// SIMATIC S7-200 SMART project (STEP 7-Micro/WIN SMART), CPU ST40

ORGANIZATION_BLOCK MAIN:OB1
TITLE=程序注释
BEGIN
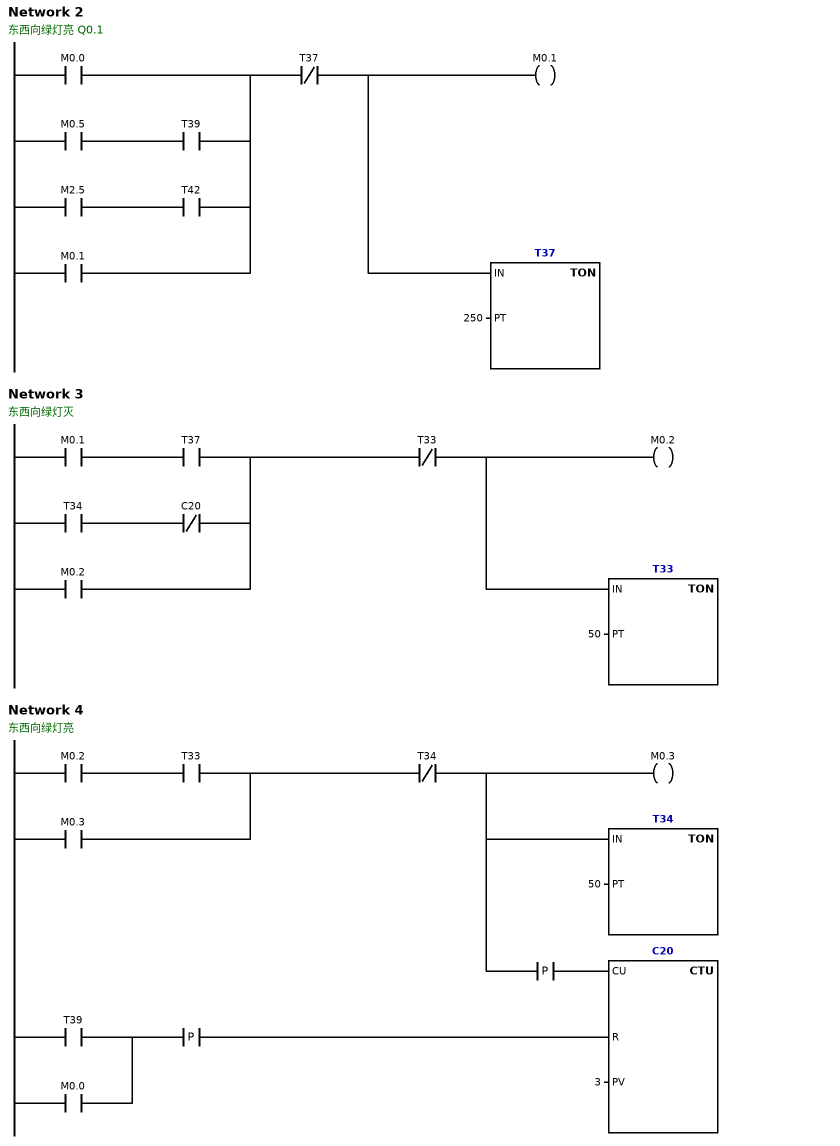
Network 2
// 东西向绿灯亮 Q0.1
// (network saved uncompiled; LAD cells follow)
// row 0: c0 -| |- M0.0  c1 -- v  c2 -|/|- T37 v  c3 --  c4 -( ) M0.1
// row 1: c0 -| |- M0.5  c1 -| |- T39 ^v  c2 ^v
// row 2: c0 -| |- M2.5  c1 -| |- T42 ^v  c2 ^v
// row 3: c0 -| |- M0.1  c1 -- ^  c2 ^  c3 --  c4 [TON T37 IN:=power@row3, PT:=250]
// row 4: c4 [box]
Network 3
// 东西向绿灯灭
// (network saved uncompiled; LAD cells follow)
// row 0: c0 -| |- M0.1  c1 -| |- T37 v  c2 --  c3 -|/|- T33 v  c4 --  c5 -( ) M0.2
// row 1: c0 -| |- T34  c1 -|/|- C20 ^v  c3 ^v
// row 2: c0 -| |- M0.2  c1 -- ^  c3 ^  c4 --  c5 [TON T33 IN:=power@row2, PT:=50]
// row 3: c5 [box]
Network 4
// 东西向绿灯亮
// (network saved uncompiled; LAD cells follow)
// row 0: c0 -| |- M0.2  c1 -| |- T33 v  c2 --  c3 -|/|- T34 v  c4 --  c5 -( ) M0.3
// row 1: c0 -| |- M0.3  c1 -- ^  c3 ^v  c4 --  c5 [TON T34 IN:=power@row1, PT:=50]
// row 2: c3 ^v  c5 [box]
// row 3: c3 ^  c4 -|P|-  c5 [CTU C20 CU:=power@row3, R:=power@row4, PV:=3]
// row 4: c0 -| |- T39 v  c1 -|P|-  c2 --  c3 --  c4 --  c5 [box]
// row 5: c0 -| |- M0.0 ^  c5 [box]
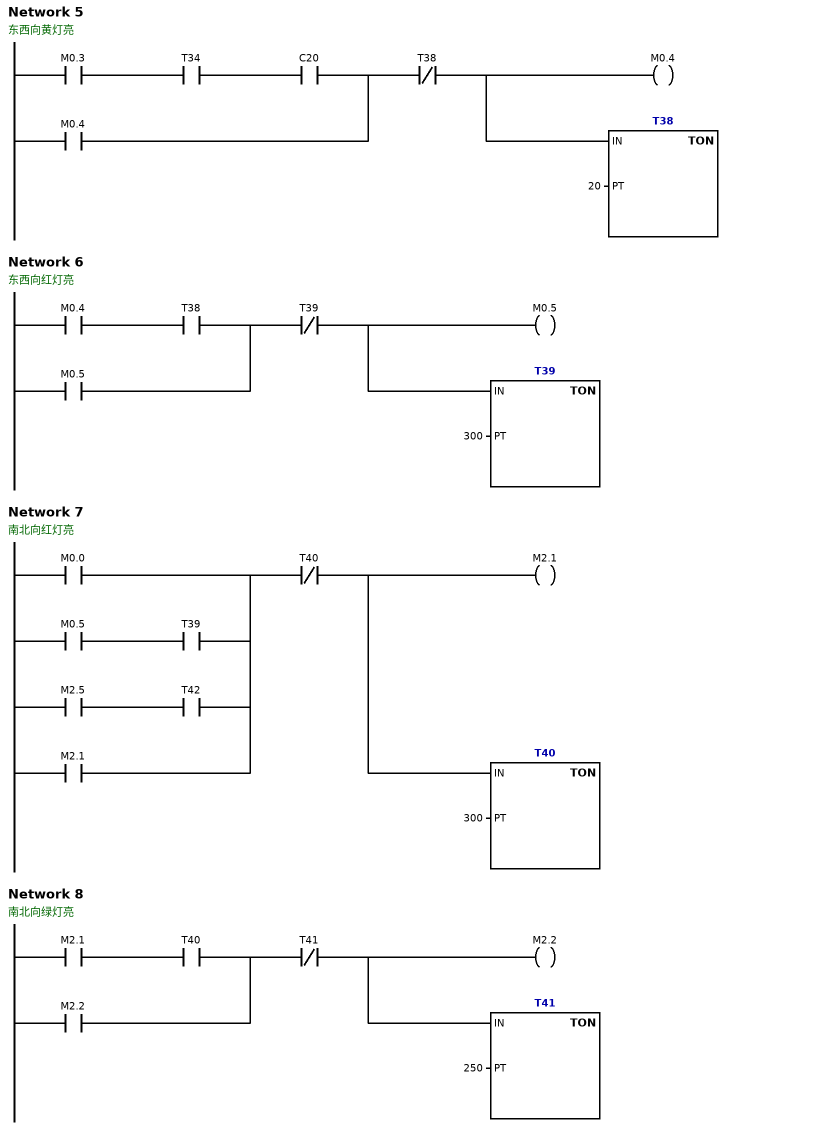
Network 5
// 东西向黄灯亮
// (network saved uncompiled; LAD cells follow)
// row 0: c0 -| |- M0.3  c1 -| |- T34  c2 -| |- C20 v  c3 -|/|- T38 v  c4 --  c5 -( ) M0.4
// row 1: c0 -| |- M0.4  c1 --  c2 -- ^  c3 ^  c4 --  c5 [TON T38 IN:=power@row1, PT:=20]
// row 2: c5 [box]
Network 6
// 东西向红灯亮
// (network saved uncompiled; LAD cells follow)
// row 0: c0 -| |- M0.4  c1 -| |- T38 v  c2 -|/|- T39 v  c3 --  c4 -( ) M0.5
// row 1: c0 -| |- M0.5  c1 -- ^  c2 ^  c3 --  c4 [TON T39 IN:=power@row1, PT:=300]
// row 2: c4 [box]
Network 7
// 南北向红灯亮
// (network saved uncompiled; LAD cells follow)
// row 0: c0 -| |- M0.0  c1 -- v  c2 -|/|- T40 v  c3 --  c4 -( ) M2.1
// row 1: c0 -| |- M0.5  c1 -| |- T39 ^v  c2 ^v
// row 2: c0 -| |- M2.5  c1 -| |- T42 ^v  c2 ^v
// row 3: c0 -| |- M2.1  c1 -- ^  c2 ^  c3 --  c4 [TON T40 IN:=power@row3, PT:=300]
// row 4: c4 [box]
Network 8
// 南北向绿灯亮
// (network saved uncompiled; LAD cells follow)
// row 0: c0 -| |- M2.1  c1 -| |- T40 v  c2 -|/|- T41 v  c3 --  c4 -( ) M2.2
// row 1: c0 -| |- M2.2  c1 -- ^  c2 ^  c3 --  c4 [TON T41 IN:=power@row1, PT:=250]
// row 2: c4 [box]
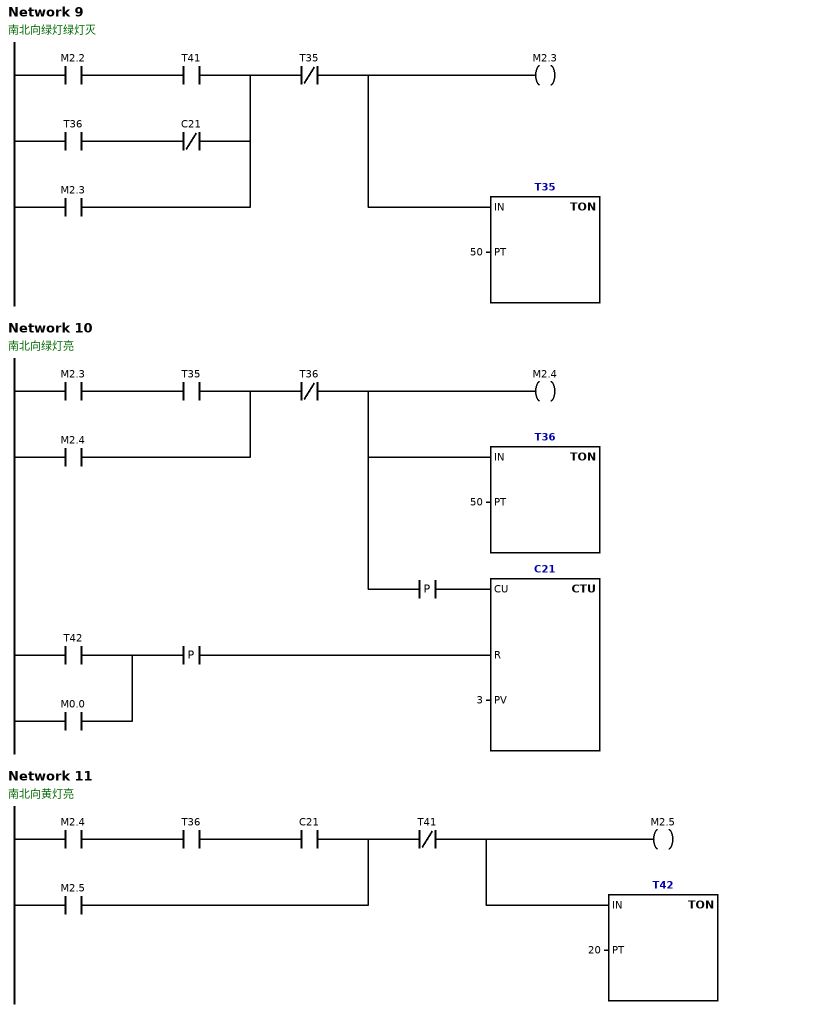
Network 9
// 南北向绿灯绿灯灭
// (network saved uncompiled; LAD cells follow)
// row 0: c0 -| |- M2.2  c1 -| |- T41 v  c2 -|/|- T35 v  c3 --  c4 -( ) M2.3
// row 1: c0 -| |- T36  c1 -|/|- C21 ^v  c2 ^v
// row 2: c0 -| |- M2.3  c1 -- ^  c2 ^  c3 --  c4 [TON T35 IN:=power@row2, PT:=50]
// row 3: c4 [box]
Network 10
// 南北向绿灯亮
// (network saved uncompiled; LAD cells follow)
// row 0: c0 -| |- M2.3  c1 -| |- T35 v  c2 -|/|- T36 v  c3 --  c4 -( ) M2.4
// row 1: c0 -| |- M2.4  c1 -- ^  c2 ^v  c3 --  c4 [TON T36 IN:=power@row1, PT:=50]
// row 2: c2 ^v  c4 [box]
// row 3: c2 ^  c3 -|P|-  c4 [CTU C21 CU:=power@row3, R:=power@row4, PV:=3]
// row 4: c0 -| |- T42 v  c1 -|P|-  c2 --  c3 --  c4 [box]
// row 5: c0 -| |- M0.0 ^  c4 [box]
Network 11
// 南北向黄灯亮
// (network saved uncompiled; LAD cells follow)
// row 0: c0 -| |- M2.4  c1 -| |- T36  c2 -| |- C21 v  c3 -|/|- T41 v  c4 --  c5 -( ) M2.5
// row 1: c0 -| |- M2.5  c1 --  c2 -- ^  c3 ^  c4 --  c5 [TON T42 IN:=power@row1, PT:=20]
// row 2: c5 [box]
END_ORGANIZATION_BLOCK
